Yaskawa INFORM job: BATMAN_2STR2.JBI

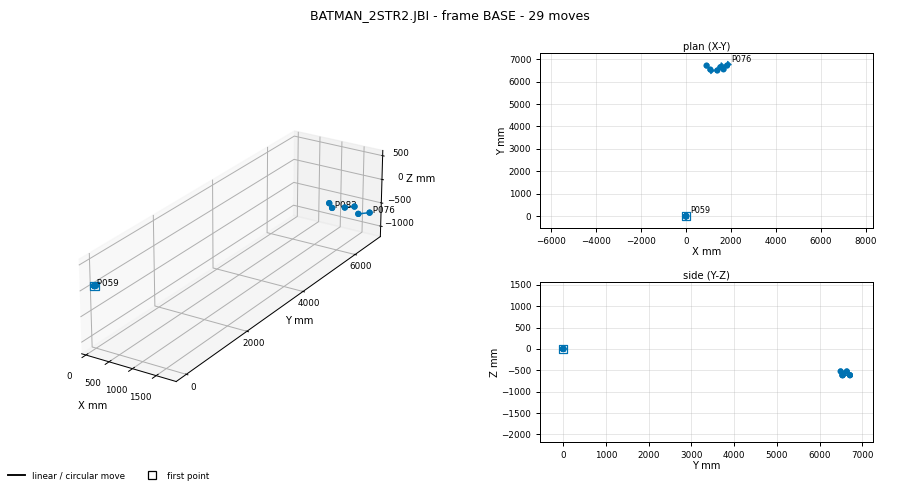
[picture p0: tool path of BATMAN_2STR2.JBI in frame BASE, 29 of 158 moves have a stored position in this frame; points joined in program order, loops and branches not executed]
/JOB
//NAME BATMAN_2STR2
///FOLDERNAME KRIS-SCIANA
//POS
///NPOS 87,87,0,38,0,0
///TOOL 0
///POSTYPE PULSE
///PULSE
C00000=-31537,-23580,-27047,-7382,83440,5380
C00001=4439,-80271,-60487,-2542,78839,17882
C00002=4909,-71742,-52465,-2581,78299,18054
C00003=4909,-71408,-51607,-2583,77943,18062
C00004=4003,-76097,-55806,-2516,78090,17746
C00005=-11747,-85634,-59902,-1317,75336,12362
C00006=-17222,-85079,-58279,-879,74547,10476
C00007=-17222,-84654,-57378,-879,74209,10479
C00008=-32420,-92461,-63354,368,73826,5218
C00009=-38310,-89326,-60200,854,73541,3171
C00010=-38411,-87974,-57554,866,72613,3131
C00011=-52965,-92159,-62746,2025,73914,-1900
C00012=-61358,-85477,-59160,2650,75381,-4774
C00013=-61358,-84056,-56150,2662,74255,-4796
C00014=-75499,-78505,-56919,3580,78174,-9561
C00015=-83067,-69095,-51058,4078,79716,-12122
C00016=-83067,-68831,-50352,4082,79419,-12132
C00017=-88580,-62756,-47818,4387,81267,-13958
C00018=-88580,-62447,-46923,4391,80875,-13971
C00019=-86164,-73606,-62214,4226,84415,-13027
C00020=-57917,-54425,-46980,-17076,96075,38866
C00021=-60111,-48306,-36516,-17002,92082,38079
C00022=-60111,-47805,-34954,-16989,91408,38172
C00023=-57173,-66532,-47658,-16705,90283,39362
C00024=-59200,-81912,-52939,-16900,85405,39315
C00025=-59200,-81575,-52247,-16904,85163,39349
C00026=-59200,-87444,-65004,-16885,89797,38712
C00027=-77293,-91319,-66542,-18032,84923,33018
C00028=-78815,-89111,-63875,-18097,84100,32600
C00029=-78815,-88680,-62940,-18106,83761,32651
C00030=-77659,-104533,-72577,-18129,81907,33338
C00031=-85944,-119702,-73803,-18852,73386,31718
C00032=-85944,-119035,-72855,-18874,73158,31754
C00033=-85944,-127357,-84566,-18634,75940,31313
C00034=-151728,-156665,-91033,10961,48688,-27461
C00035=-147386,-144150,-78835,9995,47122,-25843
C00036=-147386,-143392,-78018,10012,47009,-25856
C00037=-159688,-136539,-80417,12242,53478,-30103
C00038=-159864,-114758,-72700,11428,59817,-29460
C00039=-159864,-114128,-71743,11458,59558,-29486
C00040=-178833,-117408,-76536,14786,63793,-36172
C00041=-185982,-109235,-68028,15950,64108,-38812
C00042=-185982,-105259,-61796,16193,62382,-39063
C00043=-185982,-104478,-60574,16241,62044,-39113
C00044=-187292,-95250,-61496,15751,67410,-38841
C00045=-183818,-69704,-47887,14832,71357,-37047
C00046=-183818,-69315,-46950,14862,70992,-37094
C00047=-189068,-79923,-59995,15373,74458,-38558
C00048=-240783,-66651,-54673,5271,85755,-800
C00049=-221621,-57378,-44513,1208,77777,5604
C00050=-221621,-57331,-44364,1208,77711,5603
C00051=-221621,-56958,-43225,1210,77201,5598
C00052=-209855,-66411,-50910,-154,76995,9661
C00053=-204224,-60156,-45596,-810,76973,11605
C00054=-204224,-59837,-44664,-810,76563,11609
C00055=-190935,-64439,-49542,-2326,77463,16192
C00056=-187139,-58560,-45852,-2740,78333,17483
C00057=-187139,-58268,-44945,-2744,77925,17491
C00058=-175859,-58305,-47275,-3933,79806,21323
C00059=-173058,-51684,-42116,-4205,80175,22273
C00060=-173058,-51401,-41141,-4209,79721,22288
C00061=-163443,-46154,-39855,-5122,82181,25494
C00062=-164371,-42092,-35572,-5042,81576,25199
C00063=-164371,-41888,-34799,-5046,81206,25215
C00064=-152450,-34721,-33700,-6075,85024,29123
C00065=-152482,-28705,-27482,-6076,84290,29147
C00066=-152482,-28524,-26647,-6078,83872,29168
C00067=-149914,-24320,-24570,-6281,84946,29990
C00068=-149914,-24092,-23472,-6285,84391,30019
C00069=-149914,-25418,-31483,-6271,88614,29809
C00070=-211398,-85777,-67952,36,77534,9131
C00071=-220860,-59615,-47506,1127,78466,5876
C00072=-149914,-25418,-31483,-6271,88614,29809
C00073=-120676,-126644,-99384,-8179,81117,40244
C00074=4439,-80271,-60487,-2542,78839,17882
C00075=4965,-73716,-54196,-2585,78353,18072
C00076=-88570,-67702,-56464,4362,84042,-13858
C00077=-72474,-62815,-55247,-1455,87461,40265
C00078=-73182,-62032,-50393,-1435,84864,40051
C00079=-40588,-107108,-69894,-14776,86568,45594
C00080=-66697,-109240,-70557,-17651,80780,37350
C00081=-61032,-155504,-83571,-18589,65779,39418
C00082=-7538,-136917,-80960,-26310,62251,16305
C00083=-57429,-139298,-79120,-15077,53225,10516
C00084=-59881,-144372,-70175,-16489,44985,10894
C00085=-106253,-185325,-93876,-3450,33474,-8250
C00086=-22771,-70378,-68211,4350,89881,-13656
BC00000=150411,908787,897158
BC00001=227289,910067,536239
BC00002=227289,910067,536239
BC00003=227289,910067,536239
BC00004=227288,910066,536236
BC00005=227288,910066,536236
BC00006=227288,910066,536236
BC00007=227288,910066,536236
BC00008=227288,910066,536236
BC00009=227288,910066,536236
BC00010=227288,910066,536236
BC00011=227288,910066,536236
BC00012=227288,910066,536236
BC00013=227288,910066,536236
BC00014=227288,910066,536236
BC00015=227288,910066,536236
BC00016=227288,910066,536236
BC00017=227288,910066,536236
BC00018=227288,910066,536236
BC00019=227288,910066,536234
BC00020=227288,910065,536231
BC00021=226103,910475,539411
BC00022=226103,910475,539411
BC00023=226103,910475,539411
BC00024=226103,910475,539411
BC00025=226103,910475,539411
BC00026=226103,910475,539411
BC00027=226103,910475,539411
BC00028=226103,910475,539411
BC00029=226103,910475,539411
BC00030=226103,910475,539411
BC00031=226103,910475,539411
BC00032=226103,910475,539411
BC00033=226103,910475,539411
BC00034=226103,910475,539411
BC00035=226103,910475,539411
BC00036=226103,910475,539411
BC00037=226103,910475,539411
BC00038=226103,910475,539411
BC00039=226103,910475,539411
BC00040=226103,910475,539411
BC00041=226103,910475,539411
BC00042=226103,910475,539411
BC00043=226103,910475,539411
BC00044=226103,910475,539411
BC00045=226103,910475,539411
BC00046=226103,910475,539411
BC00047=226103,910475,539411
BC00048=227288,910066,536234
BC00049=227288,872031,536234
BC00050=227288,872031,536234
BC00051=227288,872031,536234
BC00052=227288,872031,536231
BC00053=227288,872031,536231
BC00054=227288,872031,536231
BC00055=227288,872031,536231
BC00056=227288,872031,536231
BC00057=227288,872031,536231
BC00058=227288,872031,536231
BC00059=227288,872032,536229
BC00060=227288,872032,536229
BC00061=227288,872032,536229
BC00062=227288,872032,536229
BC00063=227288,872032,536229
BC00064=227288,872032,536229
BC00065=227288,872032,536229
BC00066=227288,872032,536229
BC00067=227288,872032,536229
BC00068=227288,872032,536229
BC00069=227288,872032,536229
BC00070=227288,872032,536229
BC00071=227288,872032,536229
BC00072=227288,872032,536229
BC00073=227288,872032,536229
BC00074=227289,910067,536239
BC00075=227289,910067,536239
BC00076=227289,910067,536239
BC00077=227289,910067,536239
BC00078=227289,910067,536239
BC00079=229734,933470,547726
BC00080=229734,933470,547726
BC00081=230424,940075,550968
BC00082=134457,940075,550968
BC00083=135032,941238,551539
BC00084=135032,941238,551539
BC00085=135031,941237,551536
BC00086=135575,734603,897757
///POSTYPE BASE
///RECTAN
///RCONF 0,0,0,0,0,0,0,0,0,0,0,0,0,0,0,0,0,0,0,0,0,0,0,0
P00059=0.483,-0.984,-2.888,0.0000,0.0000,0.0000
P00060=2.327,-2.514,-2.692,0.0000,0.0000,0.0000
P00061=1.575,-3.405,-0.752,0.0000,0.0000,0.0000
P00062=-0.135,-0.848,-1.706,0.0000,0.0000,0.0000
P00063=0.036,-0.654,-3.005,0.0000,0.0000,0.0000
P00064=-0.056,-0.423,-1.596,0.0000,0.0000,0.0000
P00065=-5.731,-1.657,0.588,0.0000,0.0000,0.0000
P00070=0.003,2.805,-1.116,0.0000,0.0000,0.0000
P00071=2.716,0.070,1.352,0.0000,0.0000,0.0000
P00072=1.041,-0.003,-0.797,0.0000,0.0000,0.0000
P00073=-0.961,5.319,-6.157,0.0000,0.0000,0.0000
P00074=1.123,1.944,-5.914,0.0000,0.0000,0.0000
///RCONF 0,1,0,0,0,0,0,0,0,0,0,0,0,0,0,0,0,0,0,0,0,0,0,0
P00075=-1.802,0.025,1.546,0.0000,0.0000,0.0000
///RCONF 0,0,0,0,0,0,0,0,0,0,0,0,0,0,0,0,0,0,0,0,0,0,0,0
P00076=1830.475,6713.589,-615.047,-10.0281,37.5073,-56.2412
P00077=1670.673,6544.317,-616.315,-10.0497,37.5473,-56.2807
P00078=1529.727,6638.522,-525.778,-10.0474,37.5483,-56.2737
P00079=1392.721,6493.935,-525.116,-10.0441,37.5324,-56.2705
P00080=-3.893,-3.240,-0.208,0.0000,0.0000,0.0000
P00081=19.486,11.347,1.262,0.0000,0.0000,0.0000
P00082=1084.422,6532.900,-616.641,-10.0181,37.5185,-126.4483
P00083=916.889,6710.405,-616.123,-10.0077,37.5340,-126.4421
P00087=-17.000,22.000,-3.000,0.0000,0.0000,0.0000
P00088=-2.376,0.094,2.453,0.0000,0.0000,0.0000
P00089=5.697,-3.100,-1.263,0.0000,0.0000,0.0000
P00090=0.184,3.539,2.293,0.0000,0.0000,0.0000
P00091=-0.109,0.052,-0.075,0.0000,0.0000,0.0000
P00092=12.000,9.000,-4.000,0.0000,0.0000,0.0000
P00093=-12.000,-12.000,-3.000,0.0000,0.0000,0.0000
P00094=10.000,-10.000,-3.000,0.0000,0.0000,0.0000
P00095=-3.945,4.918,-0.177,0.0000,0.0000,0.0000
P00096=-0.633,5.398,-3.809,0.0000,0.0000,0.0000
P00108=0.000,0.000,-3.000,0.0000,0.0000,0.0000
P00109=4.000,4.000,-1.000,-10.0000,10.0000,-30.0000
P00110=13.000,-10.000,-3.000,0.0000,0.0000,0.0000
///RCONF 0,0,0,0,1,0,0,0,0,0,0,0,0,0,0,0,0,0,0,0,0,0,0,0
P00123=0.398,-92.365,-0.154,0.0099,0.0024,-0.0079
///RCONF 0,0,0,0,0,0,0,0,0,0,0,0,0,0,0,0,0,0,0,0,0,0,0,0
P00125=0.000,0.000,2.400,0.0000,0.0000,0.0000
P00126=-50.000,0.000,0.000,0.0000,0.0000,0.0000
P00127=50.000,0.000,0.000,0.0000,0.0000,0.0000
//INST
///DATE 2024/07/31 08:53
///COMM NOWY SEARCH
///ATTR SC,RW
///GROUP1 RB1,BS1
NOP
SFTOF
MOVJ C00000 BC00000 VJ=60.00
MOVJ C00001 BC00001 VJ=60.00
'POMIAR PRAWA STRONA
'1
MOVL C00002 BC00002 V=166.7
MOVL C00003 BC00003 V=16.7 PL=0 SRCH RIN#(1)=ON T=1.00 DIS=20.0
TIMER T=0.20
IMOV P125 V=13.3 PL=0
TIMER T=0.20
IMOV P127 V=13.3 PL=0 SRCH RIN#(1)=ON DIS=20.0
TIMER T=0.20
GETS PX070 $PX001
TIMER T=0.10
MOVJ C00004 BC00004 VJ=15.00
MOVJ C00005 BC00005 VJ=15.00
'2
MOVL C00006 BC00006 V=50.0
MOVL C00007 BC00007 V=16.7 PL=0 SRCH RIN#(1)=ON T=1.00 DIS=20.0
TIMER T=0.20
IMOV P125 V=13.3 PL=0
TIMER T=0.20
IMOV P127 V=13.3 PL=0 SRCH RIN#(1)=ON DIS=20.0
TIMER T=0.20
GETS PX071 $PX001
TIMER T=0.10
MOVJ C00008 BC00008 VJ=15.00
'3
MOVL C00009 BC00009 V=50.0
MOVL C00010 BC00010 V=16.7 PL=0 SRCH RIN#(1)=ON T=1.00 DIS=20.0
TIMER T=0.20
IMOV P125 V=13.3 PL=0
TIMER T=0.20
IMOV P127 V=13.3 PL=0 SRCH RIN#(1)=ON DIS=20.0
TIMER T=0.20
GETS PX072 $PX001
TIMER T=0.10
MOVJ C00011 BC00011 VJ=15.00
'4
MOVL C00012 BC00012 V=50.0
MOVL C00013 BC00013 V=16.7 PL=0 SRCH RIN#(1)=ON T=1.00 DIS=20.0
TIMER T=0.20
IMOV P125 V=13.3 PL=0
TIMER T=0.20
IMOV P127 V=13.3 PL=0 SRCH RIN#(1)=ON DIS=20.0
TIMER T=0.20
GETS PX073 $PX001
TIMER T=0.10
MOVJ C00014 BC00014 VJ=15.00
'5
MOVL C00015 BC00015 V=50.0
MOVL C00016 BC00016 V=16.7 PL=0 SRCH RIN#(1)=ON T=1.00 DIS=20.0
TIMER T=0.20
IMOV P125 V=13.3 PL=0
TIMER T=0.20
IMOV P127 V=13.3 PL=0 SRCH RIN#(1)=ON DIS=20.0
TIMER T=0.20
GETS PX074 $PX001
TIMER T=0.10
MOVL C00017 BC00017 V=50.0
MOVL C00018 BC00018 V=16.7 PL=0 SRCH RIN#(1)=ON T=1.00 DIS=20.0
TIMER T=0.20
IMOV P125 V=13.3 PL=0
TIMER T=0.20
IMOV P127 V=13.3 PL=0 SRCH RIN#(1)=ON DIS=20.0
TIMER T=0.20
GETS PX075 $PX001
TIMER T=0.10
MOVJ C00019 BC00019 VJ=15.00
MOVJ C00020 BC00020 VJ=30.00
'POMIAR BATMAN
MOVL C00021 BC00021 V=166.7
MOVL C00022 BC00022 V=16.7 PL=0 SRCH RIN#(1)=ON T=1.00 DIS=20.0
TIMER T=0.20
IMOV P125 V=13.3 PL=0
TIMER T=0.20
IMOV P123 V=13.3 PL=0 SRCH RIN#(1)=ON DIS=20.0
TIMER T=0.20
GETS PX076 $PX001
TIMER T=0.10
MOVJ C00023 BC00023 VJ=30.00
MOVL C00024 BC00024 V=166.7
MOVL C00025 BC00025 V=16.7 PL=0 SRCH RIN#(1)=ON T=1.00 DIS=20.0
TIMER T=0.20
IMOV P125 V=13.3 PL=0
TIMER T=0.20
IMOV P123 V=13.3 PL=0 SRCH RIN#(1)=ON DIS=20.0
TIMER T=0.20
GETS PX077 $PX001
TIMER T=0.10
MOVJ C00026 BC00026 VJ=30.00
MOVJ C00027 BC00027 VJ=30.00
MOVL C00028 BC00028 V=166.7
MOVL C00029 BC00029 V=16.7 PL=0 SRCH RIN#(1)=ON T=1.00 DIS=20.0
TIMER T=0.20
IMOV P125 V=13.3 PL=0
TIMER T=0.20
IMOV P123 V=13.3 PL=0 SRCH RIN#(1)=ON DIS=20.0
TIMER T=0.20
GETS PX078 $PX001
TIMER T=0.10
MOVJ C00030 BC00030 VJ=30.00
MOVL C00031 BC00031 V=166.7
MOVL C00032 BC00032 V=16.7 PL=0 SRCH RIN#(1)=ON T=1.00 DIS=20.0
TIMER T=0.20
IMOV P125 V=13.3 PL=0
TIMER T=0.20
IMOV P123 V=13.3 PL=0 SRCH RIN#(1)=ON DIS=20.0
TIMER T=0.20
GETS PX079 $PX001
TIMER T=0.10
MOVJ C00033 BC00033 VJ=30.00
MOVJ C00034 BC00034 VJ=30.00
MOVL C00035 BC00035 V=166.7
MOVL C00036 BC00036 V=16.7 PL=0 SRCH RIN#(1)=ON T=1.00 DIS=20.0
TIMER T=0.20
IMOV P125 V=13.3 PL=0
TIMER T=0.20
IMOV P123 V=13.3 PL=0 SRCH RIN#(1)=ON DIS=20.0
TIMER T=0.20
GETS PX080 $PX001
TIMER T=0.10
MOVJ C00037 BC00037 VJ=30.00
MOVL C00038 BC00038 V=166.7
MOVL C00039 BC00039 V=16.7 PL=0 SRCH RIN#(1)=ON T=1.00 DIS=20.0
TIMER T=0.20
IMOV P125 V=13.3 PL=0
TIMER T=0.20
IMOV P123 V=13.3 PL=0 SRCH RIN#(1)=ON DIS=20.0
TIMER T=0.20
GETS PX081 $PX001
TIMER T=0.10
MOVJ C00040 BC00040 VJ=30.00
MOVJ C00041 BC00041 VJ=30.00
MOVL C00042 BC00042 V=166.7
MOVL C00043 BC00043 V=16.7 PL=0 SRCH RIN#(1)=ON T=1.00 DIS=20.0
TIMER T=0.20
IMOV P125 V=13.3 PL=0
TIMER T=0.20
IMOV P123 V=13.3 PL=0 SRCH RIN#(1)=ON DIS=20.0
TIMER T=0.20
GETS PX082 $PX001
TIMER T=0.10
MOVJ C00044 BC00044 VJ=30.00
MOVL C00045 BC00045 V=166.7
MOVL C00046 BC00046 V=16.7 PL=0 SRCH RIN#(1)=ON T=1.00 DIS=20.0
TIMER T=0.20
IMOV P125 V=13.3 PL=0
TIMER T=0.20
IMOV P123 V=13.3 PL=0 SRCH RIN#(1)=ON DIS=20.0
TIMER T=0.20
GETS PX083 $PX001
TIMER T=0.10
MOVJ C00047 BC00047 VJ=30.00
'KONIEC POMIAR BATMAN 1STR
SFTOF
MOVJ C00048 BC00048 VJ=50.00
SFTOF
MOVJ C00049 BC00049 VJ=15.00
'1
MOVL C00050 BC00050 V=166.7
MOVL C00051 BC00051 V=16.7 PL=0 SRCH RIN#(1)=ON T=1.00 DIS=20.0
TIMER T=0.20
IMOV P125 V=13.3 PL=0
TIMER T=0.20
IMOV P126 V=13.3 PL=0 SRCH RIN#(1)=ON DIS=20.0
TIMER T=0.20
GETS PX059 $PX001
TIMER T=0.10
MOVJ C00052 BC00052 VJ=15.00
MOVL C00053 BC00053 V=166.7
MOVL C00054 BC00054 V=16.7 PL=0 SRCH RIN#(1)=ON T=1.00 DIS=20.0
TIMER T=0.20
IMOV P125 V=13.3 PL=0
TIMER T=0.20
IMOV P126 V=13.3 PL=0 SRCH RIN#(1)=ON DIS=20.0
TIMER T=0.20
GETS PX060 $PX001
TIMER T=0.10
MOVJ C00055 BC00055 VJ=50.00
'2
MOVL C00056 BC00056 V=50.0
MOVL C00057 BC00057 V=16.7 PL=0 SRCH RIN#(1)=ON T=1.00 DIS=30.0
TIMER T=0.20
IMOV P125 V=13.3 PL=0
TIMER T=0.20
IMOV P126 V=13.3 PL=0 SRCH RIN#(1)=ON DIS=20.0
TIMER T=0.20
GETS PX061 $PX001
TIMER T=0.10
MOVJ C00058 BC00058 VJ=50.00
'3
MOVL C00059 BC00059 V=50.0
MOVL C00060 BC00060 V=16.7 PL=0 SRCH RIN#(1)=ON T=1.00 DIS=30.0
TIMER T=0.20
IMOV P125 V=13.3 PL=0
TIMER T=0.20
IMOV P126 V=13.3 PL=0 SRCH RIN#(1)=ON DIS=20.0
TIMER T=0.20
GETS PX062 $PX001
TIMER T=0.10
MOVJ C00061 BC00061 VJ=50.00
'4
MOVL C00062 BC00062 V=50.0
MOVL C00063 BC00063 V=16.7 PL=0 SRCH RIN#(1)=ON T=1.00 DIS=30.0
TIMER T=0.20
IMOV P125 V=13.3 PL=0
TIMER T=0.20
IMOV P126 V=13.3 PL=0 SRCH RIN#(1)=ON DIS=20.0
TIMER T=0.20
GETS PX063 $PX001
TIMER T=0.10
MOVJ C00064 BC00064 VJ=15.00
'5
MOVL C00065 BC00065 V=50.0
MOVL C00066 BC00066 V=16.7 PL=0 SRCH RIN#(1)=ON T=1.00 DIS=20.0
TIMER T=0.20
IMOV P125 V=13.3 PL=0
TIMER T=0.20
IMOV P126 V=13.3 PL=0 SRCH RIN#(1)=ON DIS=20.0
TIMER T=0.20
GETS PX064 $PX001
TIMER T=0.10
MOVL C00067 BC00067 V=50.0
MOVL C00068 BC00068 V=16.7 PL=0 SRCH RIN#(1)=ON T=1.00 DIS=20.0
TIMER T=0.20
IMOV P125 V=13.3 PL=0
TIMER T=0.20
IMOV P126 V=13.3 PL=0 SRCH RIN#(1)=ON DIS=20.0
TIMER T=0.20
GETS PX065 $PX001
TIMER T=0.10
MOVJ C00069 BC00069 VJ=15.00
'********
'********
'********
MOVJ C00070 BC00070 VJ=15.00
MOVL C00071 BC00071 V=333.3
MACRO1 MJ#(0) ARGF7
SFTOF
SFTON P095
MOVL P059 V=83.3
ARCON
MOVL P060 V=10.8
MOVL P061 V=10.8
ARCON
MOVL P062 V=10.8
MOVL P063 V=10.8
MOVL P064 V=10.8
SFTOF
SFTON P109
MOVL P065 V=10.8
ARCOF
MOVJ C00072 BC00072 VJ=15.00
SFTOF
MOVJ C00073 BC00073 VJ=15.00
MOVJ C00074 BC00074 VJ=40.00
SFTON P096
MOVJ C00075 BC00075 VJ=15.00
MOVL P070 V=83.3
ARCON
MOVL P071 V=10.8
MOVL P072 V=10.8
MOVL P073 V=10.8
MOVL P074 V=10.8
SFTOF
SFTON P110
MOVL P075 V=10.8
ARCOF
SFTOF
MOVJ C00076 BC00076 VJ=15.00
MOVJ C00077 BC00077 VJ=30.00
'START SPAWANIE BATMAN
MOVJ C00078 BC00078 VJ=30.00
SFTON P090
MOVL P076 V=83.3
SFTOF
ARCON
SFTON P108
ARCON
MOVL P076 V=10.8
MOVL P077 V=10.8
SFTOF
SFTON P091
MOVL P077 V=10.8
ARCOF
SFTOF
MOVJ C00079 BC00079 VJ=30.00
MOVJ C00080 BC00080 VJ=30.00
SFTON P092
MOVL P078 V=83.3
ARCON
SFTOF
SFTON P108
MOVL P078 V=10.8
MOVL P079 V=10.8
SFTOF
SFTON P093
MOVL P079 V=10.8
ARCOF
SFTOF
MOVJ C00081 BC00081 VJ=30.00
MOVJ C00082 BC00082 VJ=30.00
SFTON P094
MOVL P080 V=83.3
SFTOF
ARCON
SFTON P108
MOVL P080 V=10.8
MOVL P081 V=10.8
SFTOF
SFTON P087
MOVL P081 V=10.8
SFTOF
ARCOF
MOVJ C00083 BC00083 VJ=30.00
MOVJ C00084 BC00084 VJ=30.00
SFTON P088
MOVL P082 V=83.3
SFTOF
ARCON
SFTON P108
MOVL P082 V=10.8
MOVL P083 V=10.8
SFTOF
SFTON P089
MOVL P083 V=10.8
SFTOF
ARCOF
MOVJ C00085 BC00085 VJ=30.00
MOVJ C00086 BC00086 VJ=100.00
CALL JOB:ONLY_CUT_KM_NEW_SCIANA
END
